	hmi_graphic_object_status_init(
        object_name         		:= CONCAT(prc_path, '_hmi_in_position_waterfall_off_hgos'),
        process             		:= prc,
        CONVERSION_this             := hmi_in_position_waterfall_off_hgos);	
	
	hmi_graphic_object_status_init(
        object_name         		:= CONCAT(prc_path, '_hmi_in_position_accumulator_depth_on_hgos'),
        process             		:= prc,
        CONVERSION_this             := hmi_in_position_accumulator_depth_on_hgos);	
	
	hmi_graphic_object_status_init(
        object_name         		:= CONCAT(prc_path, '_hmi_in_position_accumulator_depth_off_hgos'),
        process             		:= prc,
        CONVERSION_this             := hmi_in_position_accumulator_depth_off_hgos);	
	
	hmi_graphic_object_status_init(
        object_name         		:= CONCAT(prc_path, '_hmi_in_position_accumulator_conv_depth_on_hgos'),
        process             		:= prc,
        CONVERSION_this             := hmi_in_position_accumulator_conv_depth_on_hgos);	
	
	hmi_graphic_object_status_init(
        object_name         		:= CONCAT(prc_path, '_hmi_in_position_accumulator_conv_depth_off_hgos'),
        process             		:= prc,
        CONVERSION_this             := hmi_in_position_accumulator_conv_depth_off_hgos);	
	hmi_graphic_object_status_init(
        object_name         		:= CONCAT(prc_path, '_hmi_in_position_top_rail_os_width_on_hgos'),
        process             		:= prc,
        CONVERSION_this             := hmi_in_position_top_rail_os_width_on_hgos);	
	
	hmi_graphic_object_status_init(
        object_name         		:= CONCAT(prc_path, '_hmi_in_position_top_rail_os_width_off_hgos'),
        process             		:= prc,
        CONVERSION_this             := hmi_in_position_top_rail_os_width_off_hgos);	
	hmi_graphic_object_status_init(
        object_name         		:= CONCAT(prc_path, '_hmi_in_position_top_rail_ls_width_on_hgos'),
        process             		:= prc,
        CONVERSION_this             := hmi_in_position_top_rail_ls_width_on_hgos);	
	
	hmi_graphic_object_status_init(
        object_name         		:= CONCAT(prc_path, '_hmi_in_position_top_rail_ls_width_off_hgos'),
        process             		:= prc,
        CONVERSION_this             := hmi_in_position_top_rail_ls_width_off_hgos);	
	hmi_graphic_object_status_init(
        object_name         		:= CONCAT(prc_path, '_hmi_in_position_top_rail_depth_on_hgos'),
        process             		:= prc,
        CONVERSION_this             := hmi_in_position_top_rail_depth_on_hgos);	
	
	hmi_graphic_object_status_init(
        object_name         		:= CONCAT(prc_path, '_hmi_in_position_top_rail_depth_off_hgos'),
        process             		:= prc,
        CONVERSION_this             := hmi_in_position_top_rail_depth_off_hgos);	
	hmi_graphic_object_status_init(
        object_name         		:= CONCAT(prc_path, '_hmi_in_position_discharge_os_depth_on_hgos'),
        process             		:= prc,
        CONVERSION_this             := hmi_in_position_discharge_os_depth_on_hgos);	
	
	hmi_graphic_object_status_init(
        object_name         		:= CONCAT(prc_path, '_hmi_in_position_discharge_os_depth_off_hgos'),
        process             		:= prc,
        CONVERSION_this             := hmi_in_position_discharge_os_depth_off_hgos);	
	
	
//HMI graphic object status for machine is ready and enabled for visiblity of read and write button  on the RFID setup screen
	hmi_graphic_object_status_init(
        object_name         		:= CONCAT(prc_path, '_hmi_machine_ready_and_enable_hgos'),
        process             		:= prc,
        CONVERSION_this             := hmi_machine_ready_and_enable_hgos);	

		
	filter_init(
		object_name					:= CONCAT(prc_path, '_horn_on_filter'),
		delay_off_on				:= horn_on_time,
		delay_on_off				:= horn_off_time,
		process						:= prc,
		CONVERSION_this				:= horn_on_filter);
		
	
END_IF

IF objects_running()
THEN
	process_cycle(prc);
	
	command_button_cycle(hmi_toggle_cbtn);
	command_button_cycle(manual_empty_cbtn);
	command_button_cycle(RFID_Setup_read_cbtn);
	command_button_cycle(RFID_Setup_write_cbtn);
	command_button_cycle(brand_change_request_cbtn);
	command_button_cycle(navigate_to_accU_popup_cbtn);
	
	motorization_conditioner_cycle(all_in_position_motcond);
	motorization_conditioner_cycle(eoat_rfid_checked_motcond);
	motorization_conditioner_cycle(loader_pusher_rfid_checked_motcond);
	motorization_conditioner_cycle(loader_plate_rfid_checked_motcond);
	
	digital_check_cycle(stop_machine_for_change_parts_dchk);
	
	filter_cycle(accU_axis_moving_horn_on, horn_on_filter);
END_IF
END_ACTION

ACTION _read_process_image:
command_button_led_set_status(
	status				:= HMI_OBJECT_STATUS_ON, 		
	CONVERSION_this		:= brand_change_request_cbtn);

command_button_led_set_status(
	status				:= HMI_OBJECT_STATUS_ON, 		
	CONVERSION_this		:= navigate_to_accU_popup_cbtn);

brand_change_request_dvr := command_button_is_pressed(brand_change_request_cbtn);
navigate_to_accU_popup_dvr := command_button_is_pressed(navigate_to_accU_popup_cbtn);
END_ACTION

ACTION _read_var_input:
;
END_ACTION

ACTION _set_runtime_properties:
IF navigate_to_accU_popup_dvr
THEN
	navigate_to_accU_popup := FALSE;
	not_in_brand_change := TRUE;
END_IF;
END_ACTION

ACTION _write_output:
;
END_ACTION

ACTION RFID:
IF RFID_reader_list_accuchange <> RFID_reader_list_accuchange_old
THEN
	RFID_Setup_read_value_string := '';
	RFID_Setup_read_value := null_byte;
	RFID_reader_list_accuchange_old := RFID_reader_list_accuchange;
ELSE
	RFID_Setup_read_value_string := BYTE_TO_STRING(RFID_Setup_read_value);
END_IF


IF csp_main_accuChange.RFID_reader_list_accuchange = LOADER_PUSHER_READER
THEN
	loader_plate_in_position := FALSE;
	case_feed_in_position := FALSE;
	closing_os_in_position := FALSE; 
	
	change_part_color := hmi_change_part_pusher_color;
	
	changeover_rfid_read_done := csp_case_loader_pusher.rfid_read_done;
	changeover_rfid_write_done := csp_case_loader_pusher.rfid_write_done;
	changeover_rfid_value := csp_case_loader_pusher.rfid_value;
	changover_rfid_read_write_running := csp_case_loader_pusher.RFID_read_write_running;
	 
	IF csp_case_loader_pusher.rfid_input_bitheader_1.CP
	THEN
		loader_in_position := TRUE;
	END_IF
	 
	
ELSIF csp_main_accuChange.RFID_reader_list_accuchange = CASE_FEED_EOAT_READER
THEN
	loader_in_position := FALSE;
	loader_plate_in_position := FALSE;
	closing_os_in_position := FALSE; 
	
	change_part_color := hmi_change_part_eoat_color;

	changeover_rfid_read_done := csp_case_feed_arm_sensors.rfid_read_done;
	changeover_rfid_write_done := csp_case_feed_arm_sensors.rfid_write_done;
	changeover_rfid_value := csp_case_feed_arm_sensors.rfid_value;
	changover_rfid_read_write_running := csp_case_feed_arm_sensors.RFID_read_write_running;
		
	IF csp_case_feed_arm_sensors.rfid_input_bitheader_1.CP
	THEN
		case_feed_in_position := TRUE;
	END_IF
		 
ELSIF csp_main_accuChange.RFID_reader_list_accuchange = LOADER_GUIDE_PLATE_READER
THEN
	loader_in_position := FALSE;
	case_feed_in_position := FALSE;
	closing_os_in_position := FALSE;
	
	change_part_color := hmi_change_part_plate_color;
	
	changeover_rfid_read_done := csp_case_loader_sensors.rfid_read_done;
	changeover_rfid_write_done := csp_case_loader_sensors.rfid_write_done;
	changeover_rfid_value := csp_case_loader_sensors.rfid_value;
	changover_rfid_read_write_running := csp_case_loader_sensors.RFID_read_write_running;
	
	IF csp_case_loader_sensors.rfid_input_bitheader_1.CP
	THEN
		loader_plate_in_position := TRUE;
	END_IF
		
ELSIF csp_main_accuChange.RFID_reader_list_accuchange = CLOSING_PADDLES_READER
THEN
	loader_in_position := FALSE;
	case_feed_in_position := FALSE;
	loader_plate_in_position := FALSE;
	
	change_part_color := hmi_change_part_paddle_color;

	changeover_rfid_read_done := csp_case_closing.rfid_read_done;
	changeover_rfid_write_done := csp_case_closing.rfid_write_done;
	changeover_rfid_value := csp_case_closing.os_rfid_value;
	changover_rfid_read_write_running := NOT csp_case_closing.rfid_read_done OR NOT csp_case_closing.rfid_write_done;

	IF 	csp_case_closing.os_rfid_input_bitheader_1.CP
		OR csp_case_closing.ls_rfid_input_bitheader_1.CP
	THEN
		closing_os_in_position := TRUE;
	END_IF
	 
END_IF
	
	

//checks all the change parts to see if the selected part is infront of the rfid reader
IF 	loader_in_position
	OR
	case_feed_in_position
	OR
	loader_plate_in_position
	OR
	closing_os_in_position
THEN
	change_part_in_position:= TRUE;
ELSE
	change_part_in_position :=FALSE;	
END_IF

	hmi_graphic_object_set_status(
        status  			:= SEL(change_part_in_position, HMI_OBJECT_STATUS_INVISIBLE, HMI_OBJECT_STATUS_ON),
        CONVERSION_this     := hmi_in_position_on_hgos);
		
	hmi_graphic_object_set_status(
        status  			:= SEL(change_part_in_position, HMI_OBJECT_STATUS_ON, HMI_OBJECT_STATUS_INVISIBLE),
        CONVERSION_this     := hmi_in_position_off_hgos);

		
		
(* READ VALUE FROM RFID TO HIM *)
IF 	command_button_get_actual_value(RFID_Setup_read_cbtn) = HMI_BUTTON_STATUS_ON
	AND machine_is_ready(csp.mch)
THEN
	RFID_read_write_status_next := READ_WRITE_STATUS_START_RFID_READ;
END_IF


IF hmi_toggle_hgos.status = HMI_OBJECT_STATUS_ON
THEN
	enable_write := TRUE;
ELSE
	enable_write := FALSE;
END_IF

(* WRITES VALUE FROM HMI TO RFID *)
IF command_button_get_actual_value(RFID_Setup_write_cbtn) = HMI_BUTTON_STATUS_ON
	AND machine_is_ready(csp.mch)
	AND enable_write
THEN
	RFID_read_write_status_next := READ_WRITE_STATUS_START_RFID_WRITE;
END_IF

(* STATE MACHINE FOR READING AND WRITING TO RFID - ONLY FOR COMMAND BUTTONS*)
CASE RFID_read_write_status OF
	(* READ LOGIC *)
	READ_WRITE_STATUS_START_RFID_READ:
	
		rfid_read_write_running := TRUE;
		RFID_read_write_status_next := READ_WRITE_STATUS_SEND_READ_COMMAND;
		
		
	READ_WRITE_STATUS_SEND_READ_COMMAND:
	
		rfid_reading := TRUE;
		IF changover_rfid_read_write_running
		THEN
			RFID_read_write_status_next := READ_WRITE_STATUS_WAIT_FOR_READ_RESULT;
		END_IF
		
		
	READ_WRITE_STATUS_WAIT_FOR_READ_RESULT:
	
		IF 	rfid_reading
			AND changeover_rfid_read_done (* BE DYNAMIC BASED ON SELECTION - AT TOP *)
		THEN
			RFID_read_write_status_next := READ_WRITE_STATUS_CHECK_READ_RESULT;
		END_IF


	READ_WRITE_STATUS_CHECK_READ_RESULT:
	
		rfid_read_write_running := FALSE;
		rfid_reading := FALSE;
		RFID_Setup_read_value := changeover_rfid_value; (* BE DYNAMIC BASED ON SELECTION - AT TOP *)
		RFID_read_write_status_next := READ_WRITE_STATUS_WAITING;
		
		
	(* WRITE LOGIC *)
	READ_WRITE_STATUS_START_RFID_WRITE:
	
		rfid_read_write_running := TRUE;
		RFID_Setup_write_value := INT_TO_BYTE(RFID_reader_brand_colors);
		RFID_read_write_status_next := READ_WRITE_STATUS_SEND_WRITE_COMMAND;
		
		
	READ_WRITE_STATUS_SEND_WRITE_COMMAND:
	
		rfid_writing := TRUE;
		IF changover_rfid_read_write_running
		THEN
			RFID_read_write_status_next := READ_WRITE_STATUS_WAIT_FOR_WRITE_SUCCESS;
		END_IF
		
		
	READ_WRITE_STATUS_WAIT_FOR_WRITE_SUCCESS:
	
		IF rfid_writing
			AND changeover_rfid_write_done
		THEN
			rfid_read_write_running := FALSE;
			rfid_writing := FALSE;
			
			RFID_read_write_status_next := READ_WRITE_STATUS_WAITING;
		END_IF
		
		
	READ_WRITE_STATUS_WRITE_TO_READ:
	
		RFID_read_write_status_next := READ_WRITE_STATUS_START_RFID_READ;
				
		
	READ_WRITE_STATUS_WAITING:
	
		rfid_read_write_running := FALSE;	
		
		
	READ_WRITE_STATUS_ERROR:
	
		;
	
	
	
END_CASE


(* ADVANCES TO NEXT STEP *)
IF 	NOT RFID_read_write_debug
	OR
	RFID_read_write_one_step	
THEN
	RFID_read_write_status := RFID_read_write_status_next;
	RFID_read_write_one_step := FALSE;
END_IF


(* Connection timeout *)
IF	RFID_read_write_running
	AND NOT RFID_read_write_debug
THEN
	IF	timer_is_expired(RFID_read_write_tmr)
	THEN
		process_message_set(1, RFID_read_write_status, 0, RFID_read_write_error_msg);
	END_IF
ELSE
	timer_restart(10000, RFID_read_write_tmr);
END_IF
END_ACTION

END_PROGRAM

(* stored: Version 1.1.0.1, ProductVersion 3.1.4024.3
   POU csp_main_accuChange: Id {1368eecb-a803-49a7-ac9f-b9d3a373ac43}, SpecialFunc None
   Action _brand_colors: Id {dd0372cf-f1be-4b96-8eda-76ca410426b4}
   Action _handle_messages: Id {c55e7901-8c0d-409f-84ed-ca350ea22cb8}
   Action _handle_process_test: Id {6507f061-b02a-40c7-95f8-f76cf2189969}
   Action _hmi_management: Id {03365f4c-775c-4441-ba53-6fd533380dca}
   Action _in_position: Id {7ef95837-13e5-487a-b11c-cef9cdd681c5}
   Action _mode_manager: Id {2ca4eff0-aefd-4cbd-ba4a-f5b5b3acdc67}
   Action _object_manager: Id {46144055-5ff3-4453-b079-2b65d85071d9}
   Action _read_process_image: Id {c667b6b8-6d39-442e-b85c-343f521a5e5a}
   Action _read_var_input: Id {8d7d3f4c-63a2-4817-be6b-58697720ecc2}
   Action _set_runtime_properties: Id {93f5f2c7-06fa-4d9e-975b-d08223a20116}
   Action _write_output: Id {001cfdd0-67a5-4388-a497-31ac62587a99}
   Action RFID: Id {22b906b3-21ee-4eda-9877-a710b421bbd1} *)
